// TIA Portal V20 export
DATA_BLOCK "instFB_MCDDataTransfer"   // DB
TITLE = MCD Data Transfer instance DB
{ S7_Optimized_Access := 'TRUE' }
// iDB for FB_MCDDataTransfer — publishes ScaraArm3D.AxesData.A[i].{Position,Velocity} to GDB_MCDData for NX MCD viewport
// stored: InstanceOfName FB_MCDDataTransfer, InstanceOfType FB
"FB_MCDDataTransfer"
BEGIN
END_DATA_BLOCK
